(* CODESYS project PRO_JSON 1.0.0.13.library
   Version: 1.0.0.13
   Title: PRO JSON
   Author: TVM
   DocFormat: reStructuredText
   Placeholder: PRO_JSON
   Company: Pro Electric
   DefaultNamespace: PRO_JSON

Project tree, tasks and I/O mapping:
  libraries: Standard, 3.5.15.0 (System); StringUtils, 3.5.15.0 (System); SysMem, 3.5.12.0 (System)
  00000000-0000-0000-0000-000000000000|D:\Dropbox\Pro Electric\Codesys Libraries Development\Pro Electric\COPYING.txt
  00000000-0000-0000-0000-000000000000|D:\Dropbox\Pro Electric\Codesys Libraries Development\Pro Electric\GPL COPYRIGHT.txt
  COPYING
  Data Types/
    data type ASCII
    data type JSONNAMEVALUE
    data type JSONVALUETYPE
    function block JSONVAR [ST]: AsString, Boolean, CharString, FB_Init, Integer, Null, Number, ApplicationLevel, Size, ValueType, VarName, AsDateTime, Init
    data type JSONVARNAME
  Examples/
    data type EXAMPLEJSONSTRUCT
    data type EXAMPLEJSONSTRUCT_1
    program ExampleJSON_PRG [ST]
    function block EXAMPLE_FB [ST]
    program Test_ArrayOfStruct_PRG [ST]
    program Test_Array_PRG [ST]
    program Test_NestedStruct_PRG [ST]
    program Test_SingleVar_PRG [ST]
    program Test_Struct_PRG [ST]
    data type ARRAYOFSTRUCT
    data type JSONSTRUCT
    data type JSONSTRUCT_1
  Functions/
    function CLEANSTRING [ST]
    function ISBOOLEAN [ST]
    function ISNUMBER [ST]
    function block JSON_TO_STRUCT [ST]: CloseArray, CloseObject, Comma, ErrorHandler, Name, OpenArray, OpenObject, Value
    function REAL_TO_STRING_X [ST]
    function SPLIT_VARNAME [ST]
    function block STRUCT_TO_JSON [ST]: CloseArray, CloseObject, CreateArray, CreateName, CreateObject, CreateValue, ErrorHandler, Init
    function ISINTEGER [ST]
    function JSONVALUE_TO_STRING [ST]
    function STRING_TO_JSONVALUE [ST]
    function MATCH_NAMES [ST]
  GPL_COPYRIGHT
  global variables GPL_JSON
  program Notes [ST]
*)

// Data Types/ASCII
(*
| Author: Tim Van Meppelen, Pro Electric Inc.
| timv@proelectric.com
| Date: Nov 2, 2018
| enumeration of all ascii characters
*)
TYPE ASCII :
//ASCII table character definitions
(
	NULL:=			0,
 	SOH:= 			1,
 	STX:=           2,
 	ETX:=           3,
 	EOT:=           4,
 	ENQ:=           5,
 	ACK:=           6,
 	BEL:=           7,
 	BS:=            8,
 	HT:=            9,
 	LF:=            10,
 	VT:=            11,
 	FF:=            12,
 	CR:=            13,
 	SO:=            14,
 	SI:=            15,
 	DLE:=           16,
 	DC1:=           17,
 	DC2:=           18,
 	DC3:=           19,
 	DC4:=           20,
 	NAK:=           21,
 	SYN:=           22,
 	ETB:=           23,
 	CAN:=           24,
 	EM:=            25,
 	SUB_:=			26,
 	ESC:=           27,
 	FS:=            28,
 	GS:=            29,
 	RS:=            30,
 	US:=            31,
	SPACE:=			32,
	BANG:=			33,
	DOUBLE_QUOTE:=	34,
	HASH:=			35,
	DOLLAR:=		36,
	PERCENT:=		37,
	AMPERSAND:=		38,
	SINGLE_QUOTE:=	39,
	OPEN_PAREN:=	40,
	CLOSE_PAREN:=	41,
	STAR:=			42,
	PLUS:=			43,
	COMMA:=			44,
	MINUS:=			45,
	DOT:=			46,	
	SLASH:=			47,
	NUMBER_0:=		48,
	NUMBER_1:=		49,
	NUMBER_2:=		50,
	NUMBER_3:=		51,
	NUMBER_4:=		52,
	NUMBER_5:=		53,
	NUMBER_6:=		54,
	NUMBER_7:=		55,
	NUMBER_8:=		56,
	NUMBER_9:=		57,
	COLON:=			58,	
	SEMICOLON:=		59,
	LESS_THAN:=		60,
	EQUALS:=		61,
	GREATER_THAN:=	62,
	QUESTION:=		63,
	AT_SIGN:=		64,
	UPPERCASE_A:=	65,
	UPPERCASE_B:=	66,
	UPPERCASE_C:=	67,
	UPPERCASE_D:=	68,
	UPPERCASE_E:=	69,
	UPPERCASE_F:=	70,
	UPPERCASE_G:=	71,
	UPPERCASE_H:=	72,
	UPPERCASE_I:=	73,
	UPPERCASE_J:=	74,
	UPPERCASE_K:=	75,
	UPPERCASE_L:=	76,
	UPPERCASE_M:=	77,
	UPPERCASE_N:=	78,
	UPPERCASE_O:=	79,
	UPPERCASE_P:=	80,
	UPPERCASE_Q:=	81,
	UPPERCASE_R:=	82,
	UPPERCASE_S:=	83,
	UPPERCASE_T:=	84,
	UPPERCASE_U:=	85,
	UPPERCASE_V:=	86,
	UPPERCASE_W:=	87,
	UPPERCASE_X:=	88,
	UPPERCASE_Y:=	89,
	UPPERCASE_Z:=	90,
	OPEN_BRACKET:=	91,
	BACKSLASH:=		92,
	CLOSE_BRACKET:=	93,	
	CARET:=			94,
	UNDERSCORE:=	95,
	BACKQUOTE:=		96,
	LOWERCASE_A:=	97,
	LOWERCASE_B:=	98,
	LOWERCASE_C:=	99,
	LOWERCASE_D:=	100,
	LOWERCASE_E:=	101,
	LOWERCASE_F:=	102,
	LOWERCASE_G:=	103,
	LOWERCASE_H:=	104,
	LOWERCASE_I:=	105,
	LOWERCASE_J:=	106,
	LOWERCASE_K:=	107,
	LOWERCASE_L:=	108,
	LOWERCASE_M:=	109,
	LOWERCASE_N:=	110,
	LOWERCASE_O:=	111,
	LOWERCASE_P:=	112,
	LOWERCASE_Q:=	113,
	LOWERCASE_R:=	114,
	LOWERCASE_S:=	115,
	LOWERCASE_T:=	116,
	LOWERCASE_U:=	117,
	LOWERCASE_V:=	118,
	LOWERCASE_W:=	119,
	LOWERCASE_X:=	120,
	LOWERCASE_Y:=	121,
	LOWERCASE_Z:=	122,
	OPEN_BRACE:=	123,
	PIPE:=			124,
	CLOSE_BRACE:=	125,
	TILDE:=			126,
	DEL:=			127
) BYTE;
END_TYPE

// Data Types/JSONNAMEVALUE
(*
| Author: Tim Van Meppelen, Pro Electric Inc.
| timv@proelectric.com
| Date: Nov 2, 2018
| name : value pair
*)
TYPE JSONNAMEVALUE :
STRUCT
	Name:			STRING(GPL_JSON.MAX_NAME_SIZE);		//name of the object at this level
	Value:			STRING(GPL_JSON.MAX_VALUE_SIZE);	//value of the object at this level
	ArrayIndex:		UINT;	//array index of the object at this level
	IsArray:		BOOL;
END_STRUCT
END_TYPE

// Data Types/JSONVALUETYPE
(*
| Author: Tim Van Meppelen, Pro Electric Inc.
| timv@proelectric.com
| Date: Nov 2, 2018
| enumeration of all json types
| NOTE: JSON standard is somewhat ambiguous with number types, so integer and floating point numbers are separate types in this library
*)
TYPE JSONVALUETYPE :
(
	json_string,	//local var is type STRING
	json_number,	//local var is REAL
	json_integer,	//local var is DINT
	json_boolean,	//local var is BOOL
	json_null,		//local var is type null
	json_array,		//object is an array
	json_object		//object is another object (nested objects)
);
END_TYPE

// Data Types/JSONVARNAME
(*
| Author: Tim Van Meppelen, Pro Electric Inc.
| timv@proelectric.com
| Date: Nov 2, 2018
| variable name structure, used with JSONVAR
*)
TYPE JSONVARNAME :
STRUCT
	Name:			STRING(GPL_JSON.MAX_NAME_SIZE);	//name of this variable or object
	ArrayIndex:		UINT;			//array index of the object at this level
	NewObject:		BOOL;			//first variable of a new object
	EndObject:		BOOL;			//last variable of an object
	NewArray:		BOOL;			//first variable of a new array
	EndArray:		BOOL;			//last variable of an array
END_STRUCT
END_TYPE

// Examples/EXAMPLEJSONSTRUCT
(*
| Author: Tim Van Meppelen, Pro Electric Inc.
| timv@proelectric.com
| Date: Jan 31, 2020
| example of a struct of json variables
*)
TYPE EXAMPLEJSONSTRUCT :
STRUCT
	var1:		JSONVAR;
	var2:		JSONVAR;
	var3:		JSONVAR;
	obj:		EXAMPLEJSONSTRUCT_1;
	arrayobj:	ARRAY[1..3] OF JSONVAR;
END_STRUCT
END_TYPE

// Examples/EXAMPLEJSONSTRUCT_1
(*
| Author: Tim Van Meppelen, Pro Electric Inc.
| timv@proelectric.com
| Date: Jan 31, 2020
| example of a struct of json variables
*)
TYPE EXAMPLEJSONSTRUCT_1 :
STRUCT
	var4:		JSONVAR;
	var5:		JSONVAR;
	var6:		JSONVAR;
	var7:		ARRAY[1..3] OF JSONVAR;
END_STRUCT
END_TYPE

// Examples/ARRAYOFSTRUCT
TYPE ARRAYOFSTRUCT :
STRUCT
	arr:			ARRAY[1..4] OF  JSONSTRUCT;
END_STRUCT
END_TYPE

// Examples/JSONSTRUCT
TYPE JSONSTRUCT :
STRUCT
	obj1:		JSONVAR;
	_obj2:		JSONVAR;
	obj3:		JSONVAR;
END_STRUCT
END_TYPE

// Examples/JSONSTRUCT_1
TYPE JSONSTRUCT_1 :
STRUCT
	obj1:		JSONVAR;
	obj2:		JSONVAR;
	obj3:		JSONVAR;
	nest:		JSONSTRUCT;
END_STRUCT
END_TYPE

// GPL_JSON
(*
| Author: Tim Van Meppelen, Pro Electric Inc.
| timv@proelectric.com
| Date: June 26, 2018
| Parameter list that contains limits on size of strings, arrays, etc.  Most of these variables are simply
| to limit memory usage, so they can be increased or decreased to suit the local application and controller
*)
{attribute 'qualified_only'}
VAR_GLOBAL CONSTANT
	MAX_LEVELS:					UINT:= 15;		//maximum number of nested object levels
	MAX_NAME_SIZE:				UINT:= 40;		//max string length of JSON name
	MAX_VALUE_SIZE:				UINT:= 20;		//max value size in bytes (all values are this size in memory)
	MAX_VAR_NAME:				UINT:= 200;		//maximum length of full variable name with path
	MAX_VARS:					UINT:= 1500;	//maximum number of variables in the local structure
	MAX_EXECUTION_TIME:			TIME:= T#50MS;	//maximum time for a single scan of the JSON_TO_STRUCT function block
	MAX_JSON_STRING:			UINT:= 20000;	//maximum allowable size of JSON string
	NEWLINE:					STRING(2):= '$0D$0A';	//formatting string for new line
	INDENT:						STRING(1):= '$T';	//formatting string for indentation
	IGNORE_LEADING_CHAR:		STRING(1):= '_';		//ignore first character in variable names
END_VAR

// Notes
(*
| Author: Tim Van Meppelen, Pro Electric Inc.
| timv@proelectric.com
| Date: Nov 2, 2018
| 
| Tested with 200mS cyclic task, GPL_JSON.MAX_EXECUTION_TIME=50mS
| Depending on the application and speed of the controller, these values could be changed. 
| Be aware of how much cycle time is being taken when using multiple function blocks.
| Each function block will limit its time to GPL_JSON.MAX_EXECUTION_TIME, but multiple function blocks 
| could take up more than that.  This is on the list of things that could be improved. 
| 
| JSONVAR
| FB_Init will fill in information about the variable name and structure in VarNameArray
| variable type and size are automatically determined when a value is set, either:
| 	-with the set accessor of the AsString Property, which will make a guess at the type, based on the value
| 	-with any of the set accessors of the CharString, Boolean, Integer, Number, or Null properties
| variable name is set automatically in FB_Init
| 	-variable name is the JSON name
| 	-JSON allows some object names that are not valid variable names in IEC61131, for example "type", 
| 	"3h", etc.  Workaround is to put an underscore at the beginning of the variable name.  This will
| 	match in JSON_TO_STRUCT, and STRUCT_TO_JSON will create a name without the leading underscore
| 	
| JSON_TO_STRUCT
| convert a JSON string into a local structure of JSONVAR
| Long strings can take several seconds--for example, I have tested with a string of 20kB length, and the 
| parse time is about 4 seconds.  Ensuring that the local variable structure is designed to be as close as 
| possible to the expected order of variables in the JSON string will decrease parsing time, the search loop 
| always starts with the next local variable and loops around until a match is found.
| 
| STRUCT_TO_JSON
| convert a local structure of JSONVAR to a JSON string
| .Format input will create indenting and new lines, useful for writing to a file TO DO: not tested yet
| 
| GPL_JSON
| Parameter list that contains limits on size of strings, arrays, etc.  Most of these variables are simply
| to limit memory usage, so they can be increased or decreased to suit the local application and controller
|
| NEW IDEAS
| -speed up
| -JSON_STRINGIFY function that can be called multiple times to create a JSON string from key and value string inputs
| 	-would create JSON on the fly without having to define a JSONVAR structure
| 	-could be useful for small strings, HTTP server responses, etc
|	-JSONVAR.SetValue() method with ANY input might be a more convenient way to set variable values than using properties
*)
PROGRAM Notes

END_PROGRAM

// Data Types/JSONVAR
(*
| Author: Tim Van Meppelen, Pro Electric Inc.
| timv@proelectric.com
| Date: Nov 2, 2018
| local JSON variables
| 
| for use with JSON_TO_STRUCT, STRUCT_TO_JSON
| variable type and size are automatically determined when a value is set, either:
| 
| - with the set accessor of the AsString Property, which will make a guess at the type, based on the value
| - with any of the set accessors of the CharString, Boolean, Integer, Number, or Null properties
| 
| | variable name is set automatically in FB_Init:
| 
| - variable name is the JSON name
| - JSON allows some object names that are not valid variable names in IEC61131, for example "type", "3h", etc.  
| Workaround is to put a character (default: underscore) at the beginning of the variable name.  This will match in JSON_TO_STRUCT, 
| and STRUCT_TO_JSON will create a name without the leading underscore.  Character can be changed in GPL_JSON.IGNORE_LEADING_CHAR
*)
{attribute 'pack_mode' := '4'}
{attribute 'reflection'}
{attribute 'symbol' := 'none'}
FUNCTION_BLOCK JSONVAR
VAR_INPUT
	Names:			ARRAY[1..GPL_JSON.MAX_LEVELS] OF JSONVARNAME;	//variable path as an array. [1] is variable name, [2..x] are higher level structures	
END_VAR
VAR
	{attribute 'instance-path'}{attribute 'noinit'}
	{attribute 'hide'}_VarNameFull: 		STRING(GPL_JSON.MAX_VAR_NAME);   				//JSON name uses the variable name
	{attribute 'hide'}_ValueType:			JSONVALUETYPE:= JSONVALUETYPE.json_null;		//type of variable contained in the value field, also implicity defines size of local var
	{attribute 'hide'}_InternalValue:		ARRAY[1..GPL_JSON.MAX_VALUE_SIZE+1] OF BYTE;	//value stored internally as an array of bytes
	{attribute 'hide'}_Size:				UINT;										//size of internal value in bytes, automatically determined when any of the type properties are set
	{attribute 'hide'}_ApplicationLevel:	INT;										//array position which points to the application
	{attribute 'hide'}_InitDone:			BOOL;										//save if this element/ struc ... was initialisised
END_VAR
VAR_OUTPUT
	{attribute 'symbol' := 'read'}HMIVarAsString:	STRING(GPL_JSON.MAX_VALUE_SIZE); //this output is updated every time AsString property is set, for use with external HMI through sumbol configuration
END_VAR
VAR_STAT
	{attribute 'hide'}PrevApplicationLevel:	REFERENCE TO INT;		//highest variable name in previous variable
	{attribute 'hide'}PrevNameArray:		REFERENCE TO ARRAY[1..GPL_JSON.MAX_LEVELS] OF JSONVARNAME;//path of the previous variable
END_VAR

{attribute 'monitoring':='call'}PROPERTY AsString : STRING(GPL_JSON.MAX_VALUE_SIZE)
GET
(*
| Author: Tim Van Meppelen, Pro Electric Inc.
| timv@proelectric.com
| Date: Nov 2, 2018
| get the variable value as a string
*)
AsString:= JSONVALUE_TO_STRING(THIS);
END_GET
SET
(*
| Author: Tim Van Meppelen, Pro Electric Inc.
| timv@proelectric.com
| Date: Nov 2, 2018
| set the variable value as a string
*)
VAR

END_VAR
STRING_TO_JSONVALUE(
	In_String:= AsString,
	Out_JSON:= THIS
);

HMIVarAsString:= AsString;
END_SET
END_PROPERTY

{attribute 'monitoring':='call'}PROPERTY Boolean : BOOL
GET
(*
| Author: Tim Van Meppelen, Pro Electric Inc.
| timv@proelectric.com
| Date: Nov 2, 2018
| get a a boolean variable from the internal value
*)
Boolean:= BYTE_TO_BOOL(_InternalValue[1]);
END_GET
SET
(*
| Author: Tim Van Meppelen, Pro Electric Inc.
| timv@proelectric.com
| Date: Nov 2, 2018
| this is a boolean variable, copy to internal value and set type and size
*)
_ValueType:= JSONVALUETYPE.json_boolean;
_Size:= 1;

//clear memory
SysMemSet(
	pDest:= ADR(_InternalValue), 
	udiValue:= 0, 
	udiCount:= SIZEOF(_InternalValue)
);

//put data into internal value
SysMemCpy(
	pDest:= ADR(_InternalValue), 
	pSrc:= ADR(Boolean), 
	udiCount:= _Size
);
END_SET
END_PROPERTY

{attribute 'monitoring':='call'}PROPERTY CharString : STRING(GPL_JSON.MAX_VALUE_SIZE)
GET
(*
| Author: Tim Van Meppelen, Pro Electric Inc.
| timv@proelectric.com
| Date: Nov 2, 2018
| get a string variable from the internal value
*)
VAR
	TempVar:		STRING(255);
END_VAR
SysMemCpy(
	pDest:= ADR(TempVar), 
	pSrc:= ADR(_InternalValue), 
	udiCount:= _Size+1
);
CharString:= TempVar;
END_GET
SET
(*
| Author: Tim Van Meppelen, Pro Electric Inc.
| timv@proelectric.com
| Date: Nov 2, 2018
| this is a string variable, copy to internal value and set type and size
*)
_ValueType:= JSONVALUETYPE.json_string;
_Size:= INT_TO_UINT(LEN(CharString));

//clear memory
SysMemSet(
	pDest:= ADR(_InternalValue), 
	udiValue:= 0, 
	udiCount:= SIZEOF(_InternalValue)
);

//put data into internal value
SysMemCpy(
	pDest:= ADR(_InternalValue), 
	pSrc:= ADR(CharString), 
	udiCount:= _Size+1
);
END_SET
END_PROPERTY

(*
| Author: Tim Van Meppelen, Pro Electric Inc.
| timv@proelectric.com
| Date: Nov 2, 2018
| split the variable path into an array, and determine some object characteristics
| example variable path: 'Test_M241.Test_M241.Application.TestJSON_PRG.TestStruct.var1'
*)
METHOD FB_Init : BOOL
VAR_INPUT
  bInitRetains : 		BOOL; // TRUE: the retain variables are initialized (reset warm / reset cold)
  bInCopyCode : 		BOOL;  // TRUE: the instance will be copied to the copy code afterward (online change)
END_VAR

VAR
	ArrayPosition:		UINT:= GPL_JSON.MAX_LEVELS;
	NameStringPtr:		POINTER TO ARRAY[1..GPL_JSON.MAX_VAR_NAME] OF BYTE;
	StringIndex:		INT;
	VarNameBegin:		INT;
	VarNameEnd:			INT;
	VarNameIndex:		INT;
	offset:				INT;
	startarraystr:		INT;
	endarraystr:		INT;
	varlevelindex:		INT;
	prevvarlevelindex:	INT;
	stoploop:			INT;
	startloop:			INT;
	FirstVar:			BOOL;
	i:					INT;
END_VAR
//====================GET VARIABLE NAME INTO AN ARRAY====================
NameStringPtr:= ADR(_VarNameFull);
StringIndex:= LEN(_VarNameFull);
VarNameEnd:= StringIndex;
VarNameIndex:= 1;

WHILE (StringIndex > 0) DO
	IF (NameStringPtr^[StringIndex] = ASCII.DOT) THEN
	//found a "." character
		VarNameBegin:= StringIndex + 1;
		
		(*
		//clear array string  TO DO:  IS THIS NECESSARY?
		Sysmem.SysMemSet(
			pDest:= ADR(Names[VarNameIndex]), 
			udiValue:= 0, 
			udiCount:= GPL_JSON.MAX_NAME_SIZE
		);
		*)
		//copy string between VarNameBegin and VarNameEnd
		SysMem.SysMemCpy(
			pDest:= ADR(Names[VarNameIndex]), 
			pSrc:= ADR(NameStringPtr^[VarNameBegin]), 
			udiCount:= INT_TO_UDINT((VarNameEnd - VarNameBegin)+1)
		);

		//check if this is an array, if yes then remove the array index from the variable name
		startarraystr:= FIND(STR1:= Names[VarNameIndex].Name, STR2:= '[');
		endarraystr:= FIND(STR1:= Names[VarNameIndex].Name, STR2:= ']');
		IF (startarraystr <> 0) AND (endarraystr <> 0) THEN
			Names[VarNameIndex].ArrayIndex:= STRING_TO_UINT(MID(
				STR:= Names[VarNameIndex].Name, 
				LEN:= endarraystr-startarraystr-1, 
				POS:= startarraystr+1
			));
			Names[VarNameIndex].Name:= DELETE(
				STR:= Names[VarNameIndex].Name, 
				LEN:= endarraystr-startarraystr+1, 
				POS:= startarraystr
			);
		END_IF
		
		IF (Names[VarNameIndex].Name = 'Application') THEN
		//was this the application level?	
			_ApplicationLevel:= VarNameIndex;
			EXIT;
		END_IF
	
		VarNameIndex:= VarNameIndex + 1;
		VarNameEnd:= VarNameBegin - 2;	//end of the next variable name is known, store for next loop			
		StringIndex:= VarNameBegin - 2;
	ELSE
		StringIndex:= StringIndex - 1;
	END_IF
END_WHILE

//====================JSON OBJECT CHARACTERISTICS====================
(*VAR_STAT PrevApplicationLevel and PrevNameArray are references to the last JSONVAR variable
that was worked on.  This would be the previous variable in a structure or array, but
could also be a variable contained in a completely different JSON structure.
Because it is not possible to reference the next variable in a structure (because
its FB_Init() method has not run yet), the characteristics of the last variable 
in a structure are set in the STRUCT_TO_JSON function block.*)

//First variable of a structure
IF __ISVALIDREF(PrevNameArray) THEN
//there is a valid reference to a previous variable, check the previous object
	;	(*NOTE:
		I don't know if it is possible to determine whether this variable is the beginning of a new structure
		or not.  There are so many possible combinations of variables, function blocks, and structures, and the only 
		information this program has to work with is the string which contains the path.  This string only contains
		names, and does not give any information about the type of variable, or which other variables are included
		This functionality is now contained in STRUCT_TO_JSON, which is able to determine the first and last
		variables in a structure.  There's nothing really wrong with this, except that it makes the code a bit more
		difficult to understand, as there's two locations that work on variable characteristics.*)
ELSE
//there is no valid reference to a previous variable, indicating that this is the first time FB_Init has run anywhere in the application
//therefore, this is the first variable of a new JSON object
	FirstVar:= TRUE;
END_IF

IF FirstVar THEN
//first variable of a new structure
	FOR varlevelindex:= 1 TO _ApplicationLevel-2 DO
		//every level of the first variable could be either a new object or a new array
		IF (Names[varlevelindex].ArrayIndex = 1) THEN
		//new array
			Names[varlevelindex].NewArray:= TRUE;	
		ELSIF (varlevelindex > 1) THEN
		//new object
			Names[varlevelindex].NewObject:= TRUE;
		END_IF			
	END_FOR
ELSE	
//not the first variable of a new structure
	offset:= _ApplicationLevel - PrevApplicationLevel;	//check if the variable names have shifted up or down
	IF (offset < 0) THEN
	//objects shifted down
		stoploop:= PrevApplicationLevel - 1;
		startloop:= 1;
	ELSE
	//no shift, or shift up
		stoploop:= _ApplicationLevel - 1;
		startloop:= offset + 1;
	END_IF
	FOR varlevelindex:= startloop TO stoploop DO
		prevvarlevelindex:= varlevelindex - offset;
		
		//====================End previous array====================
		IF (offset < 0) AND (varlevelindex = 1) THEN
		//if objects have shifted down, then varlevelindex-offset will never point to PrevNameArray[1]
		//the previous variable might need an array closed
			IF (PrevNameArray[1].ArrayIndex > 0) THEN
			//end array
				PrevNameArray[1].EndArray:= TRUE;
			END_IF	
		END_IF

		IF (PrevNameArray[prevvarlevelindex].ArrayIndex > 0) AND (Names[varlevelindex].Name <> PrevNameArray[prevvarlevelindex].Name) THEN
			PrevNameArray[prevvarlevelindex].EndArray:= TRUE;
		END_IF	
		
		//====================End previous object====================
		IF ((varlevelindex-offset) > 1) AND ((Names[varlevelindex].Name <> PrevNameArray[prevvarlevelindex].Name) OR (Names[varlevelindex].ArrayIndex <> PrevNameArray[prevvarlevelindex].ArrayIndex)) THEN
			PrevNameArray[prevvarlevelindex].EndObject:= TRUE;	//close previous object	
		END_IF	
		
		//====================New array====================
		IF (Names[varlevelindex].ArrayIndex = 1) AND (PrevNameArray[prevvarlevelindex].ArrayIndex = 0) THEN
			Names[varlevelindex].NewArray:= TRUE;				
		END_IF	
	
		//====================New object====================
		IF (varlevelindex > 1) AND ((NOT Names[varlevelindex].NewArray) AND (Names[varlevelindex].Name <> PrevNameArray[prevvarlevelindex].Name) OR (Names[varlevelindex].ArrayIndex <> PrevNameArray[prevvarlevelindex].ArrayIndex)) THEN
			Names[varlevelindex].NewObject:= TRUE;	//new object at this level	
		END_IF	
	END_FOR

END_IF

//set a reference to some variables for the next JSON variable
PrevNameArray REF= Names;
PrevApplicationLevel REF= _ApplicationLevel;
END_METHOD

{attribute 'monitoring':='call'}PROPERTY Integer : DINT
GET
(*
| Author: Tim Van Meppelen, Pro Electric Inc.
| timv@proelectric.com
| Date: Mar 2, 2020
| get an integer variable from the internal value
| Note: .Integer and .Number are the only two properties which do type conversion on the fly because 
| the JSON standard doesn't strictly define the difference between an integer and a floating point number
*)
VAR
	tempDINT:	DINT;
	tempREAL:	REAL;
END_VAR
CASE _ValueType OF
JSONVALUETYPE.json_number:
//internal value was stored as floating point, convert to integer
	SysMemCpy(
		pDest:= ADR(tempREAL), 
		pSrc:= ADR(_InternalValue), 
		udiCount:= 4
	);
	Integer:= REAL_TO_DINT(tempREAL);		
JSONVALUETYPE.json_integer:
//internal value was stored as integer, get the value
	SysMemCpy(
		pDest:= ADR(tempDINT), 
		pSrc:= ADR(_InternalValue), 
		udiCount:= 4
	);
	Integer:= tempDINT;
END_CASE
END_GET
SET
(*
| Author: Tim Van Meppelen, Pro Electric Inc.
| timv@proelectric.com
| Date: Nov 2, 2018
| this is a integer variable, copy to internal value and set type and size
*)
VAR
	TempVar:		DINT;
END_VAR
_ValueType:= JSONVALUETYPE.json_integer;
_Size:= 4;

//clear memory
SysMemSet(
	pDest:= ADR(_InternalValue), 
	udiValue:= 0, 
	udiCount:= SIZEOF(_InternalValue)
);

TempVar:= Integer;

//put data into internal value
SysMemCpy(
	pDest:= ADR(_InternalValue), 
	pSrc:= ADR(TempVar), 
	udiCount:= _Size
);
END_SET
END_PROPERTY

{attribute 'monitoring':='call'}PROPERTY Null : STRING(4)
GET
(*
| Author: Tim Van Meppelen, Pro Electric Inc.
| timv@proelectric.com
| Date: Nov 2, 2018
| get a null value (returned as a string, as IEC61131 has no way to represent a null value)
*)
Null:= 'null';
END_GET
SET
(*
| Author: Tim Van Meppelen, Pro Electric Inc.
| timv@proelectric.com
| Date: Nov 2, 2018
| this is a null variable, set type and size
*)
_ValueType:= JSONVALUETYPE.json_null;
_Size:= 4;
END_SET
END_PROPERTY

{attribute 'monitoring':='call'}PROPERTY Number : REAL
GET
(*
| Author: Tim Van Meppelen, Pro Electric Inc.
| timv@proelectric.com
| Date: Mar 2, 2020
| get a floating point variable from the internal value
| Note: .Integer and .Number are the only two properties which do type conversion on the fly because 
| the JSON standard doesn't strictly define the difference between an integer and a floating point number
*)
VAR
	tempDINT:	DINT;
	tempREAL:	REAL;
END_VAR
CASE _ValueType OF
JSONVALUETYPE.json_integer:
//internal value was stored as integer, convert to floating point
	SysMemCpy(
		pDest:= ADR(tempDINT), 
		pSrc:= ADR(_InternalValue), 
		udiCount:= 4
	);
	Number:= DINT_TO_REAL(tempDINT);	
	
JSONVALUETYPE.json_number:
//internal value was stored as floating point, get value
	SysMemCpy(
		pDest:= ADR(tempREAL), 
		pSrc:= ADR(_InternalValue), 
		udiCount:= 4
	);
	Number:= tempREAL;	
END_CASE
END_GET
SET
(*
| Author: Tim Van Meppelen, Pro Electric Inc.
| timv@proelectric.com
| Date: Nov 2, 2018
| this is a floating point variable, copy to internal value and set type and size
*)
_ValueType:= JSONVALUETYPE.json_number;
_Size:= 4;

//clear memory
SysMemSet(
	pDest:= ADR(_InternalValue), 
	udiValue:= 0, 
	udiCount:= SIZEOF(_InternalValue)
);

//put data into internal value
SysMemCpy(
	pDest:= ADR(_InternalValue), 
	pSrc:= ADR(Number), 
	udiCount:= _Size
);
END_SET
END_PROPERTY

{attribute 'monitoring':='call'}PROPERTY ApplicationLevel : INT
GET
(*
| Author: Tim Van Meppelen, Pro Electric Inc.
| timv@proelectric.com
| Date: Nov 2, 2018
| array position which points to the application level
*)
ApplicationLevel:= _ApplicationLevel;
END_GET
END_PROPERTY

{attribute 'monitoring':='call'}PROPERTY Size : UINT
GET
(*
| Author: Tim Van Meppelen, Pro Electric Inc.
| timv@proelectric.com
| Date: Nov 2, 2018
| size of internal value in bytes, automatically determined when any of the type properties are set
*)
Size:= _Size;
END_GET
END_PROPERTY

{attribute 'monitoring':='call'}PROPERTY ValueType : JSONVALUETYPE
GET
(*
| Author: Tim Van Meppelen, Pro Electric Inc.
| timv@proelectric.com
| Date: Nov 2, 2018
| type of variable contained in the value field, also implicity defines size of local var
*)
ValueType:= _ValueType;
END_GET
SET
_ValueType:= ValueType;
END_SET
END_PROPERTY

{attribute 'monitoring':='call'}PROPERTY VarName : STRING(GPL_JSON.MAX_VAR_NAME)
GET
(*
| Author: Tim Van Meppelen, Pro Electric Inc.
| timv@proelectric.com
| Date: Sept 16, 2019
| get the name of the variable as a string, ie.
| 'Test_M241.Test_M241.Application.TestJSON_PRG.TestStruct.var1'
*)
VarName:= _VarNameFull;
END_GET
SET
(*
| Author: Tim Van Meppelen, Pro Electric Inc.
| timv@proelectric.com
| Date: Sept 16, 2019
| 
| Manually set JSON variable name to something other than it's automatically generated name.  This should only 
| be used when the JSON string could have a changing variable name at runtime, ie. the variable name is a date 
| or a counter.  Normally, the JSON variable name is the same as the PLC variable name
| NOTE:  this cannot change the number of levels of a nested object, it is assumed that the basic structure
| remains the same, and only the names are changing
| 
| example created by FB_Init:
| _VarNameFull   'Test_M241.Application.TestJSON_PRG.TestStruct.var1'
| _VarNameArray                 [4]        [3]          [2]     [1]
| _ApplicationLevel = 2
| 
| example after runtime changes
| _VarNameFull   'TestStruct.var1'
| _VarNameArray      [2]     [1]
| _ApplicationLevel = 2
| 
| set as a string ie. 'TestStruct.var1'
| each object inside another object must be changed manually
| higher level object names must be changed in each lower level object
| program level and above are not manually adjustable at runtime ie. 'Test_M241.Application.TestJSON_PRG.'
*)
VAR
	Levels:			UINT;
	i:				INT;
END_VAR
Levels:= SPLIT_VARNAME(VarNameArray:= Names, StringIn:= VarName);

FOR i:= UINT_TO_INT(Levels) TO 1 BY -1 DO 
//recreate the var name string
	IF (i = UINT_TO_INT(Levels)) THEN
		_VarNameFull:= CONCAT(Names[i].Name,'.');
	ELSIF (i = 1) THEN
		_VarNameFull:= CONCAT(_VarNameFull, Names[i].Name);
	ELSE
		_VarNameFull:= CONCAT(_VarNameFull, Names[i].Name);
		_VarNameFull:= CONCAT(_VarNameFull, '.');
	END_IF
END_FOR
END_SET
END_PROPERTY

{attribute 'monitoring':='call'}PROPERTY AsDateTime : DT
GET
(*
| Author: Tim Van Meppelen, Pro Electric Inc.
| timv@proelectric.com
| Date: Mar 2, 2020
| get a numeric JSON variable to a DATE_AND_TIME variable
*)
CASE _ValueType OF
JSONVALUETYPE.json_number:
	AsDateTime:= REAL_TO_DT(THIS^.Number);
JSONVALUETYPE.json_integer:
	AsDateTime:= DINT_TO_DT(THIS^.Integer);
JSONVALUETYPE.json_string:
	AsDateTime:= STRING_TO_DT(THIS^.CharString);
END_CASE
END_GET
SET
(*
| Author: Tim Van Meppelen, Pro Electric Inc.
| timv@proelectric.com
| Date: Mar 2, 2020
| convert the value from DATE_AND_TIME format and set it to whatever type of variable is already configured
*)
VAR
	TempReal:	REAL;
	TempInt:	DINT;
	TempString:	STRING(255);
END_VAR
CASE _ValueType OF
JSONVALUETYPE.json_number:
	TempReal:= DT_TO_REAL(AsDateTime);
	THIS^.Number:= TempReal;
JSONVALUETYPE.json_integer:
	TempInt:= DT_TO_DINT(AsDateTime);
	THIS^.Integer:= TempInt;	
JSONVALUETYPE.json_string:
	TempString:= DT_TO_STRING(AsDateTime);
	THIS^.CharString:= TempString;
END_CASE
END_SET
END_PROPERTY

PROPERTY Init : bool
SET
_InitDone:= Init;
END_SET
GET
Init:= _InitDone;
END_GET
END_PROPERTY

END_FUNCTION_BLOCK

// Functions/JSON_TO_STRUCT
(*
| Author: Tim Van Meppelen, Pro Electric Inc.
| timv@proelectric.com
| Date: Nov 2, 2018
| Last Modified: Jan 4, 2022
| parse JSON string and place the values in a matching local structure of type JSONVAR
*)
FUNCTION_BLOCK JSON_TO_STRUCT
VAR_INPUT
	Execute:			BOOL;		//rising edge triggers parse of JSON string
	Abort:				BOOL;		//rising edge stops parsing of JSON string
	JSONString:			POINTER TO ARRAY[1..GPL_JSON.MAX_JSON_STRING] OF ASCII;	//pointer to JSON string
	JSONStringSize:		UDINT;		//size of string in bytes
	JSONVars:			POINTER TO ARRAY[1..GPL_JSON.MAX_VARS] OF JSONVAR;	//pointer to local structure made up of type JSONVAR
	NumberOfVars:		UDINT;		//number of variables in the local structure or array
END_VAR

VAR_OUTPUT
	Busy:				BOOL;		//busy parsing a string
	Done:				BOOL;		//successfully parsed the whole string with no errors
	Aborted:			BOOL;		//parsing aborted by Abort input
	Error:				BOOL;		//unexpected character detected, string not completely parsed
	ErrorPosition:		UDINT;		//character position where the unexpected character was found
	ParseTime:			TIME;		//time it took to parse the string
END_VAR

VAR
	bufferposition:		UDINT;	//current position in the string
	NameValue:			ARRAY[1..GPL_JSON.MAX_LEVELS] OF JSONNAMEVALUE;	//name:value pairs currently being worked on
	obj_level:			UINT;	//number of nested objects
	name_start:			UDINT;	//index of the beginning of a name
	name_stop:			UDINT;	//index of the end of a name
	value_start:		UDINT;	//index of the beginning of a value
	value_stop:			UDINT;	//index of the end of a value
	findname:			BOOL;	//look for name in configuration array
	foundname:			BOOL;	//found a matching local var
	i:					UDINT;	//loop indexes
	jsonvarindex:		UDINT;
	levelindex:			UINT;
	nameindex:			UINT;
	thisloopstarttime:	TIME;		//time the current loop started
	starttime:			TIME;		//time parsing started
	Execute_TRIG:		R_TRIG;
	Abort_TRIG:			R_TRIG;
	findloop:			UDINT;
	parse:				BOOL;
END_VAR

IF (JSONString = 0) OR (JSONVars = 0) OR (NumberOfVars > GPL_JSON.MAX_VARS) THEN
//Bugfix Jan 4, 2022 suggested by Stefan Dreyer, to eliminate problems with uninitialized pointers	
//can't parse string - increase CPL_JSON.MAX_VARS
	Error:= TRUE;
	RETURN;
END_IF

thisloopstarttime:= TIME();	//store the time of the beginning of this loop	

Execute_TRIG(CLK:= Execute);
Abort_TRIG(CLK:= Abort);
Done:= FALSE;
IF Execute_TRIG.Q THEN
//must see a rising edge on execute to start parsing
	starttime:= TIME();	//store the time of the beginning of execution
	parse:= TRUE;
	bufferposition:= 1;
	Busy:= TRUE;
	Aborted:= FALSE;
	
	Error:= FALSE;
	ErrorPosition:= 0;
	obj_level:= 0;
	FOR i:= 1 TO GPL_JSON.MAX_LEVELS DO
		NameValue[i].Name:= '';
		NameValue[i].Value:= '';
		NameValue[i].IsArray:= FALSE;
		NameValue[i].ArrayIndex:= 0;
	END_FOR
END_IF

IF Abort_TRIG.Q THEN
	Busy:= FALSE;
	Aborted:= TRUE;
	parse:= FALSE;
END_IF

(*====================PARSE JSON STRING====================*)
//parse the input string, and start storing values in NameValue array
WHILE parse DO
	IF (JSONString^[bufferposition] = ASCII.NULL) OR (bufferposition > JSONStringSize) THEN
	//strings are terminated with a null character
	//there might not always be a null character, for example in a network buffer that is stored as an array of bytes
		parse:= FALSE;
		Done:= TRUE;
		Busy:= FALSE;
		ParseTime:= TIME() - starttime;
		RETURN;
	END_IF	

	CASE JSONString^[bufferposition] OF 

	ASCII.DOUBLE_QUOTE:	// " name string
		Name();
		
	ASCII.OPEN_BRACE:// {, beginning of object
		OpenObject();	
		
	ASCII.CLOSE_BRACE:// }, end of object
		CloseObject();
		
	ASCII.OPEN_BRACKET:	// [, beginning of array
		OpenArray();
		
	ASCII.CLOSE_BRACKET:	// ], end of array
		CloseArray();
		
	ASCII.COLON:	// :, separator for name:value pairs
		Value();
		
	ASCII.COMMA:	// , move to next object
		Comma();
	
	ASCII.SOH..ASCII.SPACE:	// skip all control characters, including spaces
		bufferposition:= bufferposition + 1;

	ELSE
	//error, unexpected character
		ErrorHandler();
	END_CASE
	
	(*========================================LOOK FOR NAMES IN LOCAL VARIABLES========================================*)
	IF findname THEN
	//there is at least one valid name:value pair in the NameValue array--check for a match in the Config array, including nested objects
		findname:= FALSE;
		FOR findloop:= 1 TO NumberOfVars DO
		(*loop through all configured objects and look for the name that is currently being worked on in the JSON string
		Local JSON object should be as closely matched to the expected JSON string as possible, to decrease parsing time.  
		This function will eventually find all objects, but it will start looking after the previous found variable, as it 
		is assumed that that's the most likely position for the next variable*)  
			jsonvarindex:= (jsonvarindex MOD NumberOfVars) + 1;
			FOR nameindex:= 1 TO obj_level DO
			//Match name and array index.  Array index will be 0 if the current name:value is not part of an array
				IF MATCH_NAMES(JSONVars^[jsonvarindex].Names[nameindex], NameValue[obj_level-(nameindex-1)]) THEN	
					foundname:= TRUE;	//name in JSON string matches the local variable name
				ELSE
					foundname:= FALSE;	//name in JSON string does not match the local variable name, go to next name
					EXIT;
				END_IF
			END_FOR
			IF foundname THEN
				EXIT;
			END_IF
		END_FOR
	
		(*====================FOUND NAME, WRITE LOCAL VAR====================*)
		IF foundname THEN
		//local var name matches with JSON string name
			foundname:= FALSE;
			JSONVars^[jsonvarindex].AsString:= NameValue[obj_level].Value;	
		END_IF
	END_IF

	IF TIME() >= (thisloopstarttime + GPL_JSON.MAX_EXECUTION_TIME) THEN
	//this function block won't take up more than GPL_JSON.MAX_EXECUTION_TIME on one scan
	//very long strings or files could take too long to parse in one task cycle, and cause a watchdog exception
		RETURN;
	END_IF
END_WHILE

(*
| Author: Tim Van Meppelen, Pro Electric Inc.
| timv@proelectric.com
| Date: Oct 22, 2018
| end of an array
*)
METHOD PRIVATE CloseArray
NameValue[obj_level].IsArray:= FALSE;
NameValue[obj_level].ArrayIndex:= 0;
bufferposition:= bufferposition + 1;
END_METHOD

(*
| Author: Tim Van Meppelen, Pro Electric Inc.
| timv@proelectric.com
| Date: Oct 22, 2018
| end of an object, move down in the object hierarchy
*)
METHOD PRIVATE CloseObject
VAR
	shiftindex:			INT;
END_VAR
NameValue[obj_level].Name:= '';
NameValue[obj_level].Value:= '';
NameValue[obj_level].IsArray:= FALSE;
NameValue[obj_level].ArrayIndex:= 0;
obj_level:= obj_level - 1;
bufferposition:= bufferposition + 1;
END_METHOD

(*
| Author: Tim Van Meppelen, Pro Electric Inc.
| timv@proelectric.com
| Date: Oct 22, 2018
| found a comma, parse an array value, or move on to the next object	
*)
METHOD PRIVATE Comma
IF NameValue[obj_level].IsArray THEN
//if this is an array at the current object level, increment the array index
	NameValue[obj_level].ArrayIndex:= NameValue[obj_level].ArrayIndex + 1;
	Value();
ELSE
	bufferposition:= bufferposition + 1;
END_IF
END_METHOD

(*
| Author: Tim Van Meppelen, Pro Electric Inc.
| timv@proelectric.com
| Date: Oct 22, 2018
| Unexpected or invalid character found, end parsing
*)
METHOD PRIVATE ErrorHandler
parse:= FALSE;
Busy:= FALSE;
Error:= TRUE;
ErrorPosition:= bufferposition;	//return buffer position of unexpected character
END_METHOD

(*
| Author: Tim Van Meppelen, Pro Electric Inc.
| timv@proelectric.com
| Date: Oct 22, 2018
| found the first quote at the beginning of a name string,
| extract the name string and put it into the NameValue array
*)
METHOD PRIVATE Name
VAR
	namestringok:		BOOL;
	j:					UDINT;
END_VAR
name_start:= bufferposition + 1;
FOR j:= name_start TO (name_start+GPL_JSON.MAX_NAME_SIZE) DO
	IF (JSONString^[j] = ASCII.DOUBLE_QUOTE) THEN
	//find the closing quote of a name string
		name_stop:= j - 1;		//name ends at character before quote
		bufferposition:= j + 1;	//next loop can start after the quote
		namestringok:= TRUE;
		EXIT;
	END_IF
END_FOR

IF namestringok THEN
	SysMemSet(
		pDest:= ADR(NameValue[obj_level].Name), 
		udiValue:= 0, 
		udiCount:= SIZEOF(NameValue[obj_level].Name)
	);
	
	SysMemCpy(
		pDest:= ADR(NameValue[obj_level].Name), 
		pSrc:= ADR(JSONString^[name_start]), 
		udiCount:= (name_stop+1 - name_start)
	);
ELSE
	ErrorHandler();
END_IF
END_METHOD

(*
| Author: Tim Van Meppelen, Pro Electric Inc.
| timv@proelectric.com
| Date: Oct 22, 2018
| found the beginning of an array, set array definition at this object level
*)
METHOD PRIVATE OpenArray
VAR_INPUT
END_VAR
NameValue[obj_level].IsArray:= TRUE;
NameValue[obj_level].ArrayIndex:= 1;
bufferposition:= bufferposition + 1;
END_METHOD

(*
| Author: Tim Van Meppelen, Pro Electric Inc.
| timv@proelectric.com
| Date: Oct 22, 2018
| found the beginning of a new object, increment the object level
*)
METHOD PRIVATE OpenObject
VAR
	shiftindex:			INT;
END_VAR
obj_level:= obj_level + 1;	//move up a level in the object hierarchy
bufferposition:= bufferposition + 1;
END_METHOD

(*
| Author: Tim Van Meppelen, Pro Electric Inc.
| timv@proelectric.com
| Date: Oct 22, 2018
| found a ":" character, possible next characters are any combination of the following:
| { begin another object
| [ begin a new array
| " or a number or letter: value found
| after all { and [ are found, and if any were found, the next thing will be a name string
| loop through until a value is found, incrementing obj_level or array definitions as necessary
*)
METHOD PRIVATE Value
VAR
	lookforname:	BOOL;
	j:				UDINT;
	skipnext:		BOOL;
	quotedstring:	BOOL;
END_VAR
bufferposition:= bufferposition + 1;	//start searching after the ":" character

WHILE (bufferposition < JSONStringSize) DO
	CASE JSONString^[bufferposition] OF
		
	ASCII.CR:	// '$r', skip
		bufferposition := bufferposition+1;
		CONTINUE;
	ASCII.LF:	// '$n', skip
		bufferposition := bufferposition+1;
		CONTINUE;
	ASCII.SPACE:	// ' ', skip
		bufferposition := bufferposition+1;
		CONTINUE;
		
	ASCII.OPEN_BRACE:// {, beginning of new object
		OpenObject();	
		lookforname:= TRUE;
	
	ASCII.OPEN_BRACKET:	// [, beginning of new array
		OpenArray();
		
	ELSE
		IF lookforname THEN
		//a new object or array was found, and all nested objects have already been looped through, therefore this buffer position must start a new name
		//there is no value here, so exit this loop, main loop should now continue at the name, and parse its name:value pair
			EXIT;
		END_IF
		
		IF (JSONString^[bufferposition] = ASCII.DOUBLE_QUOTE) THEN
		//value starts with a quote character--quoted string
			value_start:= bufferposition + 1;	//value follows : and "
			quotedstring := TRUE;	
		ELSE
			value_start:= bufferposition;	//value immediately follows :
		END_IF

		FOR j:= value_start TO JSONStringSize DO
			IF skipnext THEN
				skipnext := FALSE;
			ELSIF (JSONString^[j] = ASCII.BACKSLASH)  THEN
				// on backslash, escape the next one
				skipnext := TRUE;
			ELSIF (JSONString^[j] = ASCII.DOUBLE_QUOTE)  THEN
			//end of value is is found at the closing quote
				value_stop:= j - 1;
				bufferposition:= j + 1;	//main loop can resume at the next character after the quote
				EXIT;
			//ELSIF ((JSONString^[j] = ASCII.COMMA) OR (JSONString^[j] = ASCII.CLOSE_BRACE) OR (JSONString^[j] = ASCII.CLOSE_BRACKET)) AND (NOT quotedstring) THEN
			(*bugfix - Dec 8, 2021 Stefan Dryer
			some strings might contain a CR/LF after the value, ahead of the closing bracket*)
			ELSIF ((JSONString^[j] = ASCII.COMMA) OR (JSONString^[j] = ASCII.CLOSE_BRACE) OR (JSONString^[j] = ASCII.CLOSE_BRACKET) OR (JSONString^[j] = ASCII.CR ) OR (JSONString^[j] = ASCII.LF )) AND NOT quotedstring THEN
			//end of value is is found at , or }, or ]
				value_stop:= j - 1;
				bufferposition:= j;	//main loop can resume at the next character after the value
				EXIT;
			END_IF
		END_FOR	
		//clear previous string
		SysMemSet(
			pDest:= ADR(NameValue[obj_level].Value), 
			udiValue:= 0, 
			udiCount:= GPL_JSON.MAX_VALUE_SIZE
		);		
		//copy buffer to temporary value as a string
		SysMemCpy(
			pDest:= ADR(NameValue[obj_level].Value), 
			pSrc:= ADR(JSONString^[value_start]), 
			udiCount:= MIN((value_stop+1) - value_start, GPL_JSON.MAX_VALUE_SIZE-1)
		);
		
		findname:= TRUE;		//there is a name:value pair in the NameValue array, check for a match with a local variable
		EXIT;
	END_CASE
END_WHILE
END_METHOD

END_FUNCTION_BLOCK

// Functions/MATCH_NAMES
(*
| Author: Tim Van Meppelen, Pro Electric Inc.
| timv@proelectric.com
| Date: May 7, 2021
| compare name in JSON string with local variable name
| match when local variable name contains a leading underscore, if present
| JSON allows some object names that are not valid variable names in IEC61131, for example "type", 
| "3h", etc.  Workaround is to put an underscore at the beginning of the variable name.
| this leading underscore can be changed or not used by modifying GPL_JSON.IGNORE_LEADING_CHAR
*)
FUNCTION MATCH_NAMES : BOOL
VAR_INPUT
	Name1:			JSONVARNAME;	//name:value in local value
	Name2:			JSONNAMEVALUE;	//name:value from JSON string
END_VAR
VAR
	LocalVarName:	STRING(GPL_JSON.MAX_NAME_SIZE);	//name stripped of leading underscore, if present
END_VAR

IF (FIND(STR1:= Name1.Name, STR2:= GPL_JSON.IGNORE_LEADING_CHAR) = 1) THEN
//leading character is present, delete it 
	LocalVarName:= DELETE(Name1.Name,1,1);
END_IF

MATCH_NAMES:= ((Name1.Name = Name2.Name OR (Name2.Name = LocalVarName))AND 
				(Name1.ArrayIndex = Name2.ArrayIndex)) ;

END_FUNCTION

// Functions/STRUCT_TO_JSON
(*
| Author: Tim Van Meppelen, Pro Electric Inc.
| timv@proelectric.com
| with thanks to these contributors:
| Stefan Dreyer github.com/stefandreyer
| Wesley Vercoutere
| Date: Nov 2, 2018
| Last Modified: Jan 4, 2022
| create a JSON string from a structure of JSONVAR types
*)
FUNCTION_BLOCK STRUCT_TO_JSON
VAR_INPUT
	Execute:			BOOL;		//rising edge triggers compose of JSON string
	Abort:				BOOL;		//rising edge stops composing a JSON string
	JSONString:			POINTER TO ARRAY[1..GPL_JSON.MAX_JSON_STRING] OF ASCII;	//pointer to JSON string
	JSONStringSize:		UDINT;		//size of string
	JSONVars:			POINTER TO ARRAY[1..GPL_JSON.MAX_VARS] OF JSONVAR;	//pointer to local structure made up of type JSONVAR
	NumberOfVars:		UINT;		//number of variables in the local structure or array
	VariableArraySize:	BOOL;		//don't write array values which are null, resulting in variable array sizes
	{info <'TO DO:  Format input not tested'>}Format:	BOOL;		//add white space and indenting to the resulting string
	MaxLevel:			INT;		//max level at which to create objects
	(*by default, STRUCT_TO_JSON will create variables starting at (Application level - 2).
	This will work for most variables and structures defined in a program.  If your variable
	or structure is contained inside a function block, or nested in function blocks, it may
	be necessary to set MaxLevel to restrict creating JSON after a certain level
	MaxLevel examples:
	Device: 4, Application: 3, Program: 2, Variable: 1
	Device.Application.TestJSON_PRG.var1, default {"var1":"value"}
	Device.Application.TestJSON_PRG.var1, set MaxLevel=2 to get {TestJSON_PRG:{"var1":"value"}}
	
	Device: 5, Application: 4, Program: 3, Function Block: 2, Variable: 1
	Device.Application.TestJSON_PRG.Test_FB.var1, set MaxLevel=1 to get {"var1":"value"}
	Device.Application.TestJSON_PRG.Test_FB.var1, set MaxLevel=2 to get {Test_FB:{"var1":"value"}}
	Device.Application.TestJSON_PRG.Test_FB.var1, set MaxLevel=3 to get {TestJSON_PRG:{Test_FB:{"var1":"value"}}} 
	*)
END_VAR

VAR_OUTPUT
	Busy:				BOOL;		//busy composing a string
	Done:				BOOL;		//successfully composed the whole string with no errors
	Aborted:			BOOL;		//compose aborted by Abort input
	Error:				BOOL;		//unexpected character detected, string not completely composed
	ErrorPosition:		UDINT;		//index of local object at which composing stopped
	ComposeTime:		TIME;		//time it took to compose the string
END_VAR

VAR
	bufferposition:		UDINT;	//current position in the string
	jsonvarindex:		UDINT;
	compose:			BOOL;	
	objectstr:			STRING(255);	//string created by current variable
	names:				ARRAY[1..GPL_JSON.MAX_LEVELS] OF JSONVARNAME;	//helper variable for names array property
	namesindex:			INT;
	i:					UINT;
	
	Execute_TRIG:		R_TRIG;
	Abort_TRIG:			R_TRIG;
	thisloopstarttime:	TIME;		//time the current loop started
	starttime:			TIME;		//time composing started
	maxlevelindex:		INT;
	closeLevel: 		INT;
	objectLevel: 		INT;
	inArray: 			BOOL;
	lastindex:			UDINT;
	InitDn:				BOOL;
END_VAR

IF (JSONString = 0) OR (JSONVars = 0) OR (NumberOfVars > GPL_JSON.MAX_VARS) THEN
//Bugfix Jan 4, 2022 suggested by Stefan Dreyer, to eliminate problems with uninitialized pointers
	Error:= TRUE;
	RETURN;
END_IF

thisloopstarttime:= TIME();	//store the time of the beginning of this loop
Done:= FALSE;
Execute_TRIG(CLK:= Execute);
Abort_TRIG(CLK:= Abort);

IF Execute_TRIG.Q THEN
//must see a rising edge on execute to start composing
	starttime:= TIME();	//store the time of the beginning of execution
	compose:= TRUE;
	Busy:= TRUE;
	Aborted:= FALSE;
	//need to init every sing struct at first time...
	lastindex:= MIN(NumberOfVars, GPL_JSON.MAX_VARS);
	IF NOT JSONVars^[1].Init THEN
		JSONVars^[1].Init := Init();
	END_IF
	
	Error:= FALSE;
	ErrorPosition:= 0;
	bufferposition:= 1;
	jsonvarindex:= 1;
	objectLevel := 0;	
	FOR i:= 1 TO GPL_JSON.MAX_LEVELS DO
	//clear names array
		names[i].Name:= '';
		names[i].ArrayIndex:= 0;
	END_FOR
	//clear previous string
	SysMemSet(
		pDest:= JSONString, 
		udiValue:= 0, 
		udiCount:= JSONStringSize
	);
END_IF

IF Abort_TRIG.Q THEN
	Busy:= FALSE;
	Aborted:= TRUE;
	compose:= FALSE;
END_IF

WHILE compose AND (jsonvarindex <= lastindex) AND (bufferposition < JSONStringSize) DO 
//loop through all variables

	names:= JSONVars^[jsonvarindex].Names;	//helper variable for name array property

	IF (jsonvarindex = 1) THEN
	//first object, no comma
		objectstr:= '{';	//new JSON string	
		IF Format THEN
			objectstr:= CONCAT(objectstr, GPL_JSON.NEWLINE);
		END_IF
	ELSE
		objectstr:= '';	//clear previous object string	
		IF NOT (VariableArraySize AND (names[1].ArrayIndex > 0) AND (JSONVars^[jsonvarindex].ValueType = JSONVALUETYPE.json_null)) THEN
		//don't write the value if the current variable is an array, and the value is null
			objectstr:= CONCAT(objectstr, ',');	//comma in between each value
			IF Format AND (names[1].ArrayIndex <= 1) THEN
			//new line after each comma, except in arrays
				objectstr:= CONCAT(objectstr, GPL_JSON.NEWLINE);	
			END_IF	
		END_IF
	END_IF

	IF (MaxLevel = 0) THEN
	//default, create all objects below the program level
		maxlevelindex:= JSONVars^[jsonvarindex].ApplicationLevel - 2;
	ELSE
	//manually defined with the MaxLevel input
		IF (jsonvarindex = 1) THEN
			maxlevelindex:= MaxLevel;
		ELSE
			maxlevelindex:= JSONVars^[jsonvarindex].ApplicationLevel - 2;	
		END_IF
	END_IF
	
	FOR namesindex:= maxlevelindex TO 1 BY -1 DO 
	//loop through all levels of an object in reverse
		//======================open new objects or arrays, or create new name:value pairs======================
		IF names[namesindex].NewArray AND (names[namesindex].ArrayIndex <= 1) THEN
		//new array at this level
			CreateName(Name:= names[namesindex].Name);
			CreateArray();
		END_IF	
		IF names[namesindex].NewObject AND (namesindex <> 1) THEN
		//new object at this level
			IF (NOT inArray) THEN
				CreateName(Name:= names[namesindex].Name);
			END_IF	
			CreateObject();		
		END_IF
		
		IF (namesindex=1) THEN
		//only write a value at level 1
			IF (names[namesindex].ArrayIndex > 0) THEN
			//array, create value only
				IF NOT (VariableArraySize AND (names[1].ArrayIndex > 0) AND (JSONVars^[jsonvarindex].ValueType = JSONVALUETYPE.json_null)) THEN
				//don't write the value if the current variable is an array, and the value is null
					CreateValue(ValueType:= JSONVars^[jsonvarindex].ValueType, Value:= JSONVars^[jsonvarindex].AsString);					
				END_IF
			ELSE
			//name:value pair
				CreateName(Name:= names[namesindex].Name);
				CreateValue(ValueType:= JSONVars^[jsonvarindex].ValueType, Value:= JSONVars^[jsonvarindex].AsString);
			END_IF
		END_IF
	END_FOR
	
	
	IF (MaxLevel = 0) THEN
	//default, close all objects below the program level
		closeLevel:= JSONVars^[jsonvarindex].ApplicationLevel - 2;
	ELSE
	//manually defined with the MaxLevel input
		IF jsonvarindex = 1 THEN
			closeLevel:= 1;
		ELSE
			closeLevel:= JSONVars^[jsonvarindex].ApplicationLevel - 2;	
		END_IF
	END_IF
	
	FOR namesindex:= 1 TO closeLevel DO 
	//start at the lowest level and count up
	//close objects or arrays if this is the last value in this object or array
		IF names[namesindex].EndObject AND (namesindex <> 1) THEN
		//close object at this level
			CloseObject();
		END_IF
		
		IF names[namesindex].EndArray THEN	
		//close array at this level
			CloseArray();	
		END_IF		
		
	END_FOR	
	
	//concatenate the temporary object string to the JSON string output
	StrConcatA(
		pstFrom:= ADR(objectstr), 
		pstTo:= ADR(JSONString^[bufferposition]), 
		iBufferSize:= UDINT_TO_INT(JSONStringSize)
	);	
	
	bufferposition:= bufferposition + DINT_TO_UDINT(LEN(objectstr));

	IF (jsonvarindex >= NumberOfVars) THEN
	//end of vars, close string
		compose:= FALSE;
		Busy:= FALSE;
		Done:= TRUE;		
		ComposeTime:= TIME() - starttime;
		JSONString^[bufferposition]:= ASCII.CLOSE_BRACE;;	//close JSON object with }
		bufferposition:= bufferposition + 1;
		JSONString^[bufferposition]:= ASCII.NULL;	//null character to end string
	END_IF
	
	IF TIME() >= (thisloopstarttime + GPL_JSON.MAX_EXECUTION_TIME) THEN
	//this function block won't take up more than GPL_JSON.MAX_EXECUTION_TIME on one scan
	//very long strings could take too long to compose in one task cycle, and cause a watchdog exception
		RETURN;
	END_IF
	
	jsonvarindex:= jsonvarindex + 1;	
END_WHILE

(*
| Author: Tim Van Meppelen, Pro Electric Inc.
| timv@proelectric.com
| Date: Oct 22, 2018
| close a JSON array
*)
METHOD PRIVATE CloseArray
objectstr:= CONCAT(objectstr, ']');

IF Format THEN
	objectstr:= CONCAT(objectstr, GPL_JSON.NEWLINE);	
END_IF

inArray := FALSE;
END_METHOD

(*
| Author: Tim Van Meppelen, Pro Electric Inc.
| timv@proelectric.com
| Date: Oct 22, 2018
| close a JSON object
*)
METHOD PRIVATE CloseObject
VAR
	indent:		INT;
END_VAR
IF Format THEN
	FOR indent:= 1 TO JSONVars^[jsonvarindex].ApplicationLevel-1 DO
		objectstr:= CONCAT(objectstr, GPL_JSON.INDENT);	
	END_FOR
END_IF

IF objectLevel > 0 THEN
	objectstr:= CONCAT(objectstr, '}');
	objectLevel := objectLevel - 1;
END_IF
END_METHOD

(*
| Author: Tim Van Meppelen, Pro Electric Inc.
| timv@proelectric.com
| Date: Oct 22, 2018
| create a new JSON array
| 
| [ ------ ------------ value ---------------- ] 
|         /                               \
| 	      \_______________ , _____________/
| 		
*)
METHOD PRIVATE CreateArray
objectstr:= CONCAT(objectstr, '[');	//opening [

inArray := TRUE;
END_METHOD

(*
| Author: Tim Van Meppelen, Pro Electric Inc.
| timv@proelectric.com
| Date: Oct 22, 2018
| create a JSON name string from a local variable of type JSONVAR
*)
METHOD PRIVATE CreateName
VAR_INPUT
	Name:	 		STRING(GPL_JSON.MAX_NAME_SIZE);
END_VAR
VAR
	indent:			INT;
	leadingpos:		INT;
END_VAR
IF Format THEN
	FOR indent:= 1 TO JSONVars^[jsonvarindex].ApplicationLevel-1 DO
		objectstr:= CONCAT(objectstr, GPL_JSON.INDENT);	
	END_FOR
END_IF

objectstr:= CONCAT(objectstr, '"');	//opening quote

leadingpos:= FIND(Name, GPL_JSON.IGNORE_LEADING_CHAR);
//if leading character is configured and present, delete it from the name
IF (leadingpos = 1) THEN
	objectstr:= CONCAT(objectstr, DELETE(Name, 1, 1));//variable name
ELSE
	objectstr:= CONCAT(objectstr, Name);//variable name
END_IF

objectstr:= CONCAT(objectstr, '":');	//closing quote and name:value separator
END_METHOD

(*
| Author: Tim Van Meppelen, Pro Electric Inc.
| timv@proelectric.com
| Date: Oct 22, 2018
| create a new JSON object
| 
| {------ "name" ------ : ----- value --------- }
|     /                                 \
| 	  \_______________ , _______________/
| 
*)
METHOD PRIVATE CreateObject
objectstr:= CONCAT(objectstr, '{');	//opening {

IF Format THEN
	objectstr:= CONCAT(objectstr, GPL_JSON.NEWLINE);
END_IF

objectLevel := objectLevel + 1;
END_METHOD

(*
| Author: Tim Van Meppelen, Pro Electric Inc.
| timv@proelectric.com
| Date: Oct 22, 2018
| create a JSON value string from a local variable of type JSONVAR
*)
METHOD PRIVATE CreateValue
VAR_INPUT
	ValueType:		JSONVALUETYPE;
	Value:			STRING(GPL_JSON.MAX_VALUE_SIZE);
END_VAR
CASE ValueType OF
//append value to object string
JSONVALUETYPE.json_number:
	objectstr:= CONCAT(objectstr, Value);
JSONVALUETYPE.json_integer:
	objectstr:= CONCAT(objectstr, Value);	
JSONVALUETYPE.json_boolean:
	objectstr:= CONCAT(objectstr, Value);
JSONVALUETYPE.json_string:
	objectstr:= CONCAT(objectstr, '"');	//opening quote
	objectstr:= CONCAT(objectstr, Value);
	objectstr:= CONCAT(objectstr, '"');	//closing quote
JSONVALUETYPE.json_null:
	objectstr:= CONCAT(objectstr, 'null');
END_CASE
END_METHOD

(*
| Author: Tim Van Meppelen, Pro Electric Inc.
| timv@proelectric.com
| Date: Oct 22, 2018
| Something went wrong, return the index of the variable where the problem was encountered
*)
METHOD PRIVATE ErrorHandler
compose:= FALSE;
Busy:= FALSE;
Error:= TRUE;
ErrorPosition:= jsonvarindex;	//return buffer position of unexpected character
RETURN;
END_METHOD

METHOD PRIVATE Init : BOOL
VAR
	varlevelindex:		INT;
END_VAR
//======================Set first and lastvariable properties======================
//characteristics of the first and last variable are not always set properly by FB_Init
FOR varlevelindex:= 1 TO JSONVars^[1].ApplicationLevel-2 DO
//every level of the first variable could be either a new object or a new array
	IF (JSONVars^[1].Names[varlevelindex].ArrayIndex = 1) THEN
	//new array at the first array object
		JSONVars^[1].Names[varlevelindex].NewArray:= TRUE;	
	ELSIF (varlevelindex > 1) OR (NumberofVars = 1) THEN
	//new object at every level, special case for single variables
		JSONVars^[1].Names[varlevelindex].NewObject:= TRUE;
	END_IF			
END_FOR

//lastindex:= MIN(NumberOfVars, GPL_JSON.MAX_VARS);
FOR varlevelindex:= 1 TO JSONVars^[lastindex].ApplicationLevel-2 DO
//close all open arrays and objects
	IF (JSONVars^[lastindex].Names[varlevelindex].ArrayIndex > 0) THEN
	//end array if an array index exists
		JSONVars^[lastindex].Names[varlevelindex].EndArray:= TRUE;	
	ELSIF (varlevelindex > 1) OR (NumberofVars = 1) THEN
	//end all objects, special case for single variables
		JSONVars^[lastindex].Names[varlevelindex].EndObject:= TRUE;
	END_IF			
END_FOR

Init:= TRUE;
END_METHOD

END_FUNCTION_BLOCK

// Functions/JSONVALUE_TO_STRING
(*
| Author: Tim Van Meppelen, Pro Electric Inc.
| timv@proelectric.com
| Date: May 4, 2021
| convert a JSON value to string
*)
FUNCTION JSONVALUE_TO_STRING : STRING
VAR_INPUT
	In_JSON:		POINTER TO JSONVAR;
END_VAR

CASE In_JSON^.ValueType OF
JSONVALUETYPE.json_null:
	JSONVALUE_TO_STRING:= 'null';
JSONVALUETYPE.json_boolean:
	IF In_JSON^.Boolean THEN
		JSONVALUE_TO_STRING:= 'true';
	ELSE
		JSONVALUE_TO_STRING:= 'false';
	END_IF
JSONVALUETYPE.json_number:
	JSONVALUE_TO_STRING:= REAL_TO_STRING_X(In_JSON^.Number);
JSONVALUETYPE.json_integer:
	JSONVALUE_TO_STRING:= DINT_TO_STRING(In_JSON^.Integer);
JSONVALUETYPE.json_string:
	JSONVALUE_TO_STRING:= In_JSON^.CharString;
END_CASE

END_FUNCTION

// Functions/REAL_TO_STRING_X
(*
| Author: Tim Van Meppelen, Pro Electric Inc.
| timv@proelectric.com
| Date: Nov 2, 2018
| Standard REAL_TO_STRING function will always add a decimal place even if the input is a whole number
| this function will drop the ".0" on the string output
*)
FUNCTION REAL_TO_STRING_X : STRING
VAR_INPUT
	In_REAL:		REAL;
END_VAR
VAR
	TempVar:		STRING;
END_VAR

TempVar:= REAL_TO_STRING(In_REAL);
IF (RIGHT(STR:= TempVar, SIZE:= 2) = '.0') THEN
	REAL_TO_STRING_X:= DELETE(STR:= TempVar, LEN:= 2, POS:= LEN(TempVar) - 1);
ELSE
	REAL_TO_STRING_X:= TempVar;
END_IF

END_FUNCTION

// Functions/STRING_TO_JSONVALUE
(*
| Author: Tim Van Meppelen, Pro Electric Inc.
| timv@proelectric.com
| Date: May 4, 2021
| Convert a string to a JSON value
*)
FUNCTION STRING_TO_JSONVALUE
VAR_INPUT
	In_String:		STRING;
	Out_JSON:		POINTER TO JSONVAR;
END_VAR
VAR
	TempBool:	BOOL;
	TempReal:	REAL;
	TempInt:	DINT;
	TempString:	STRING(255);
END_VAR

IF (Out_JSON^.ValueType = JSONVALUETYPE.json_null) THEN
//if the type is not explicitly configured, make a guess at the type
	IF ISINTEGER(ADR(In_String)) THEN
		Out_JSON^.ValueType:= JSONVALUETYPE.json_integer;
	ELSIF ISNUMBER(ADR(In_String)) THEN
		Out_JSON^.ValueType:= JSONVALUETYPE.json_number;
	ELSIF ISBOOLEAN(ADR(In_String)) THEN
		Out_JSON^.ValueType:= JSONVALUETYPE.json_boolean;
	ELSIF (In_String = 'null') THEN
		Out_JSON^.ValueType:= JSONVALUETYPE.json_null;
	ELSE
		Out_JSON^.ValueType:= JSONVALUETYPE.json_string;
	END_IF
END_IF

CASE Out_JSON^.ValueType OF
JSONVALUETYPE.json_null:
	Out_JSON^.Null:= 'null';
JSONVALUETYPE.json_boolean:
	StrToUpperA(pString:= ADR(In_String));
	IF (In_String = 'TRUE') THEN
		TempBool:= TRUE;
	ELSE
		TempBool:= FALSE;
	END_IF
	Out_JSON^.Boolean:= TempBool;
JSONVALUETYPE.json_integer:
	TempInt:= STRING_TO_DINT(In_String);
	Out_JSON^.Integer:= TempInt;	
JSONVALUETYPE.json_number:
	TempReal:= STRING_TO_REAL(In_String);
	Out_JSON^.Number:= TempReal;
JSONVALUETYPE.json_string:
	Out_JSON^.CharString:= In_String;
END_CASE

END_FUNCTION

// Functions/ISINTEGER
(*
| Author: Tim Van Meppelen, Pro Electric Inc.
| timv@proelectric.com
| Date: Mar 2, 2020
| check if a string contains an integer, allows for "-" at the beginning of the string, and no decimals
*)
FUNCTION ISINTEGER : BOOL
VAR_INPUT
	In:		POINTER TO ARRAY[1..255] OF BYTE;
END_VAR
VAR
	i:				UINT;
	founddecimal:	BOOL;
END_VAR

FOR i:= 1 TO 255 DO
	CASE In^[i] OF 	
	ASCII.NULL:
	//end of string
		EXIT;
	ASCII.MINUS:
	//only allow a "-" in the first position	
		IF (i=1) THEN
			ISINTEGER:= TRUE;
		ELSE
			ISINTEGER:= FALSE;
			EXIT;
		END_IF
	ASCII.DOT:
	//no decimal points allowed in integers
		ISINTEGER:= FALSE;
		EXIT;
	ASCII.NUMBER_0..ASCII.NUMBER_9:
		ISINTEGER:= TRUE;
	ELSE
	//all other characters are not part of numbers
		ISINTEGER:= FALSE;
		EXIT;
	END_CASE
END_FOR

END_FUNCTION

// Functions/ISNUMBER
(*
| Author: Tim Van Meppelen, Pro Electric Inc.
| timv@proelectric.com
| Date: Oct 2, 2018
| check if a string contains a valid number, allows for "-" at the beginning of the string, and one "." character
*)
FUNCTION ISNUMBER : BOOL
VAR_INPUT
	In:		POINTER TO ARRAY[1..255] OF BYTE;
END_VAR
VAR
	i:				UINT;
	founddecimal:	BOOL;
END_VAR

FOR i:= 1 TO 256 DO
	CASE In^[i] OF 	
	ASCII.NULL:
	//end of string
		RETURN;
	ASCII.MINUS:
	//only allow a "-" in the first position	
		IF (i=1) THEN
			ISNUMBER:= TRUE;
		ELSE
			ISNUMBER:= FALSE;
			RETURN;
		END_IF
	ASCII.DOT:
	//only allow one decimal point
		IF founddecimal THEN
		//already found one decimal, can't have two
			ISNUMBER:= FALSE;
			RETURN;
		ELSE
		//first decimal point found, allow one
			ISNUMBER:= TRUE;
			founddecimal:= TRUE;
		END_IF
	ASCII.NUMBER_0..ASCII.NUMBER_9:
		ISNUMBER:= TRUE;
	ELSE
	//all other characters are not part of numbers
		ISNUMBER:= FALSE;
		RETURN;
	END_CASE
END_FOR

END_FUNCTION

// Functions/ISBOOLEAN
(*
| Author: Tim Van Meppelen, Pro Electric Inc.
| timv@proelectric.com
| Date: Oct 2, 2018
| check if a string would convert to a valid boolean variable
*)
FUNCTION ISBOOLEAN : BOOL
VAR_INPUT
	In:		POINTER TO STRING(5);
END_VAR
VAR
	TempVar:	STRING(5);
END_VAR

TempVar:= In^;
StrToUpperA(pString:= ADR(TempVar));

ISBOOLEAN:= (TempVar = 'TRUE') OR (TempVar = 'FALSE');

END_FUNCTION

// Functions/SPLIT_VARNAME
(*
| Author: Tim Van Meppelen, Pro Electric Inc.
| timv@proelectric.com
| Date: June 26, 2018
| split a string into an array at the '.' character
| modified from https://forum.codesys.com/viewtopic.php?t=9889
| 'a.b.c.d' becomes an array[1]=d, [2]=c, [3]=b, [4]=a
*)
FUNCTION SPLIT_VARNAME : UINT;
VAR_INPUT
	VarNameArray:	REFERENCE TO ARRAY[1..GPL_JSON.MAX_LEVELS] OF JSONVARNAME;
	StringIn: 		STRING(GPL_JSON.MAX_VAR_NAME);	//input string
END_VAR

VAR CONSTANT
	SPLIT_CHAR : 	STRING(1):= '.';	
END_VAR

VAR
	ArraySize:			UINT:= 1;
    sShortString : 		STRING;
    iSplitLocation : 	INT;
	i:					UINT;
	TempArray:			ARRAY[1..GPL_JSON.MAX_LEVELS] OF STRING;
END_VAR

//Loop through string until there is no string left or array has hit its limits
WHILE (StrLenA(pstData:= ADR(StringIn)) > 0) DO
	//Find location of first break point
	iSplitLocation := StrFindA(
		pst1:= ADR(StringIn), 
		pst2:= ADR(SPLIT_CHAR), 
		uiSearchStart:= 1
	) - 1;
	
	//If there is no break point found then set location to size of string
	IF (iSplitLocation = -1) THEN
		iSplitLocation := DINT_TO_INT(StrLenA(pstData:= ADR(StringIn)));
	END_IF
  
	//Copy the part of the string that is needed for the parameter.
	StrMidA(
		pst:= ADR(StringIn), 
		uiInputBufferSize:= SIZEOF(StringIn), 
		iLength:= iSplitLocation, 
		iPosition:= 1, 
		pstResult:= ADR(sShortString), 
		uiResultBufferSize:= SIZEOF(sShortString)
	);

	//Make sure string is not empty before using up an array spot.
	IF (StrLenA(pstData:= ADR(sShortString)) > 0) THEN
		TempArray[ArraySize] := sShortString;
		ArraySize := ArraySize + 1;
	END_IF

	//Remove copied components from long string
	StrDeleteA(
		pby:= ADR(StringIn), 
		iLength:= (iSplitLocation + LEN(SPLIT_CHAR)), 
		iPosition:= 1
	);

	//Check to see if more parameters can fit in array. If not exit loop
	IF (ArraySize > GPL_JSON.MAX_LEVELS) THEN
		EXIT;
	END_IF 
END_WHILE

ArraySize:= ArraySize - 1;

FOR i:= 0 TO ArraySize DO
//reverse the order of the array
	VarNameArray[i+1].Name:= TempArray[ArraySize-i];	
END_FOR

SPLIT_VARNAME:= ArraySize;

END_FUNCTION

// Examples/ExampleJSON_PRG
(*
| Author: Tim Van Meppelen, Pro Electric Inc.
| timv@proelectric.com
| Date: Nov 2, 2018
| example program demonstrating JSONVAR, STRUCT_TO_JSON, AND JSON_TO_STRUCT
| 
| This example will populate a structure with values and types.  On a rising edge of ComposeJSON.Execute, 
| ComposeJSON will create a JSON string.  When ComposeJSON.Done is set, ParseJSON.Execute is set, and 
| ParseJSON will then parse that string back into a different structure.
*)
PROGRAM ExampleJSON_PRG
VAR
	LocalJSONObj:		EXAMPLEJSONSTRUCT;
	ComposeJSON:		STRUCT_TO_JSON;
	
	JSONString:			STRING(1000);

	NewJSONObj:			EXAMPLEJSONSTRUCT;	
	ParseJSON:			JSON_TO_STRUCT;
	
	CreateJSONInFB:		EXAMPLE_FB;
END_VAR

LocalJSONObj.var1.Boolean:= TRUE;
LocalJSONObj.var2.Number:= 34.8756;
LocalJSONObj.var3.CharString:= 'teststring';
LocalJSONObj.obj.var4.Number:= 22;
LocalJSONObj.obj.var5.AsString:= 'FALSE';	//JSONVAR will guess at type, in this case, boolean
LocalJSONObj.obj.var6.CharString:= 'qwer';
LocalJSONObj.obj.var7[1].Number:= 123.234;
LocalJSONObj.obj.var7[2].AsString:= '55.46';	//JSONVAR will guess at type, in this case, a number
LocalJSONObj.obj.var7[3].Number:= 985;
LocalJSONObj.arrayobj[1].Number:= 1;
LocalJSONObj.arrayobj[2].Number:= 2;
LocalJSONObj.arrayobj[3].Number:= 3;

//create a JSON string from local object
ComposeJSON(
	JSONString:= ADR(JSONString), 
	JSONStringSize:= SIZEOF(JSONString),
	JSONVars:= ADR(LocalJSONObj),
	NumberOfVars:= SIZEOF(LocalJSONObj) / SIZEOF(JSONVAR)
);

//fill another local object with values from the created JSON string
ParseJSON(
	Execute:= ComposeJSON.Done,
	JSONString:= ADR(JSONString), 
	JSONStringSize:= SIZEOF(JSONString),
	JSONVars:= ADR(NewJSONObj),
	NumberOfVars:= SIZEOF(NewJSONObj) / SIZEOF(JSONVAR)
);

CreateJSONInFB();

END_PROGRAM

// Examples/EXAMPLE_FB
(*
| Author: Tim Van Meppelen, Pro Electric Inc.
| timv@proelectric.com
| Date: Jan 31, 2020
| example of use in a function block
*)
FUNCTION_BLOCK EXAMPLE_FB
VAR_INPUT
	MaxLevel:			INT;
END_VAR
VAR_OUTPUT
	Out:				STRING(255);
END_VAR
VAR
	color_temp:			JSONVAR;
	FirstScan:			BOOL:= TRUE;
	ComposeJSON:		STRUCT_TO_JSON;
END_VAR

color_temp.CharString:= 'red';

ComposeJSON(
	JSONString:= ADR(Out), 
	JSONStringSize:= SIZEOF(Out),
	JSONVars:= ADR(color_temp),
	NumberOfVars:= SIZEOF(color_temp) / SIZEOF(JSONVAR),
	MaxLevel:= MaxLevel
);

IF FirstScan THEN
	FirstScan:= FALSE;
	ComposeJSON.Execute:= TRUE;
END_IF

END_FUNCTION_BLOCK

// Functions/CLEANSTRING
(*
| Author: Tim Van Meppelen, Pro Electric Inc.
| timv@proelectric.com
| Date: Oct 9, 2018
| strip all control characters and spaces from a string
*)
FUNCTION CLEANSTRING : BOOL
VAR_INPUT
	StringPtr:		POINTER TO ARRAY[1..MAXSTRINGLENGTH] OF BYTE;
END_VAR
VAR CONSTANT
	MAXSTRINGLENGTH:	UINT:= 2048;
END_VAR
VAR
	i:				UINT;
	j:				UINT;
END_VAR

FOR i:= 1 TO MAXSTRINGLENGTH DO
	IF (StringPtr^[i] >= 1) AND (StringPtr^[i] <= 16#20) THEN
	//match all control and white space characters, except for null, which terminates a string
		FOR j:= i TO MAXSTRINGLENGTH DO
			IF (StringPtr^[j] = ASCII.NULL) THEN
			//null character terminates string
				EXIT;
			ELSE
			//shift character array left one
				StringPtr^[j]:= StringPtr^[j+1];
			END_IF
		END_FOR
		i:= i - 1;	//run loop at same position again
	ELSIF (StringPtr^[i] = ASCII.NULL) THEN
	//found null character at the end of the string
		EXIT;
	END_IF
END_FOR

CLEANSTRING:= TRUE;

END_FUNCTION

// Examples/Test_ArrayOfStruct_PRG
PROGRAM Test_ArrayOfStruct_PRG
VAR
	FirstScan:			BOOL:= TRUE;	
	
	LocalJSONObj:		ARRAYOFSTRUCT;
	ComposeJSON:		STRUCT_TO_JSON;
	JSONString:			STRING(255);

END_VAR

IF FirstScan THEN
	FirstScan:= FALSE;
	ComposeJSON.Execute:= TRUE;
END_IF

//create a JSON string
LocalJSONObj.arr[1].obj1.Number:= 23.5;
LocalJSONObj.arr[1]._obj2.Integer:= 3;
LocalJSONObj.arr[1].obj3.Boolean:= TRUE;

LocalJSONObj.arr[2].obj1.Number:= 54.5;
LocalJSONObj.arr[2]._obj2.Number:= 7.5;
LocalJSONObj.arr[2].obj3.Boolean:= FALSE;

LocalJSONObj.arr[3].obj1.Number:= 87.1;
LocalJSONObj.arr[3]._obj2.Integer:= 88;
LocalJSONObj.arr[3].obj3.Boolean:= TRUE;

LocalJSONObj.arr[4].obj1.Boolean:= FALSE;
LocalJSONObj.arr[4]._obj2.Number:= 132.55;
LocalJSONObj.arr[4].obj3.Integer:= 3;


ComposeJSON(
	JSONString:= ADR(JSONString), 
	JSONStringSize:= SIZEOF(JSONString),
	JSONVars:= ADR(LocalJSONObj),
	NumberOfVars:= SIZEOF(LocalJSONObj) / SIZEOF(JSONVAR)
);

END_PROGRAM

// Examples/Test_Array_PRG
PROGRAM Test_Array_PRG
VAR
	FirstScan:			BOOL:= TRUE;	
	
	testarray:			ARRAY[1..20] OF JSONVAR;
	ComposeJSON:		STRUCT_TO_JSON;
	JSONString:			STRING(255);
	
	NewString:			STRING(255):= '{"new":["234","34.5","98.4","10.4","812","5","23","65","95.6","98","234","34.5","98.4","10.4","812","5","23","65","95.6","98"]}';
	ParseJSON:			JSON_TO_STRUCT;
	new:				ARRAY[1..20] OF JSONVAR;	
END_VAR

IF FirstScan THEN
	FirstScan:= FALSE;
	ComposeJSON.Execute:= TRUE;
	ParseJSON.Execute:= TRUE;
END_IF

//create a JSON string
testarray[1].Number:= 32.5;
testarray[2].Number:= 65.2;
testarray[3].Number:= 81.54;
testarray[4].Number:= 1953.523;
testarray[5].Number:= 901.5;

ComposeJSON(
	JSONString:= ADR(JSONString), 
	JSONStringSize:= SIZEOF(JSONString),
	JSONVars:= ADR(testarray),
	NumberOfVars:= SIZEOF(testarray) / SIZEOF(JSONVAR)
);




//parse a JSON string and put it into a variable
ParseJSON(
	JSONString:= ADR(NewString), 
	JSONStringSize:= SIZEOF(NewString),
	JSONVars:= ADR(new),
	NumberOfVars:= SIZEOF(new) / SIZEOF(JSONVAR)
);

END_PROGRAM

// Examples/Test_NestedStruct_PRG
PROGRAM Test_NestedStruct_PRG
VAR
	FirstScan:			BOOL:= TRUE;	
	
	LocalJSONObj:		JSONSTRUCT_1;
	ComposeJSON:		STRUCT_TO_JSON;
	JSONString:			STRING(255);
	
	NewString:			STRING(255):= '{"new":{"obj1":"234", "obj2":"34.5", "obj3":"true","nest":{"obj1":"468.5", "obj2":"197", "obj3":"this is a string"}}}';
	ParseJSON:			JSON_TO_STRUCT;
	new:				JSONSTRUCT_1;
END_VAR

IF FirstScan THEN
	FirstScan:= FALSE;
	ComposeJSON.Execute:= TRUE;
	ParseJSON.Execute:= TRUE;
END_IF

//create a JSON string
LocalJSONObj.obj1.Number:= 23.5;
LocalJSONObj.obj2.Integer:= 3;
LocalJSONObj.obj3.Boolean:= TRUE;

ComposeJSON(
	JSONString:= ADR(JSONString), 
	JSONStringSize:= SIZEOF(JSONString),
	JSONVars:= ADR(LocalJSONObj),
	NumberOfVars:= SIZEOF(LocalJSONObj) / SIZEOF(JSONVAR)
);





//parse a JSON string and put it into a variable
ParseJSON(
	JSONString:= ADR(NewString), 
	JSONStringSize:= SIZEOF(NewString),
	JSONVars:= ADR(new),
	NumberOfVars:= SIZEOF(new) / SIZEOF(JSONVAR)
);

END_PROGRAM

// Examples/Test_SingleVar_PRG
PROGRAM Test_SingleVar_PRG
VAR
	FirstScan:			BOOL:= TRUE;	
	
	colour:				JSONVAR;	
	ComposeJSON:		STRUCT_TO_JSON;
	JSONString:			STRING(255);
	
	NewString:			STRING:= '{"color":"blue"}';
	ParseJSON:			JSON_TO_STRUCT;
	color:				JSONVAR;
END_VAR

IF FirstScan THEN
	FirstScan:= FALSE;
	ComposeJSON.Execute:= TRUE;
	ParseJSON.Execute:= TRUE;
END_IF

//create a JSON string from a variable
colour.CharString:= 'blue';
ComposeJSON(
	JSONString:= ADR(JSONString), 
	JSONStringSize:= SIZEOF(JSONString),
	JSONVars:= ADR(colour),
	NumberOfVars:= SIZEOF(colour) / SIZEOF(JSONVAR)
);



//parse a JSON string and put it into a variable
ParseJSON(
	JSONString:= ADR(NewString), 
	JSONStringSize:= SIZEOF(NewString),
	JSONVars:= ADR(color),
	NumberOfVars:= SIZEOF(color) / SIZEOF(JSONVAR)
);

END_PROGRAM

// Examples/Test_Struct_PRG
PROGRAM Test_Struct_PRG
VAR
	FirstScan:			BOOL:= TRUE;	
	
	LocalJSONObj:		JSONSTRUCT;
	ComposeJSON:		STRUCT_TO_JSON;
	JSONString:			STRING(255);
	
	NewString:			STRING:= '{"new":{"obj1":"234", "_obj2":"34.5", "obj3":"true"}}';
	ParseJSON:			JSON_TO_STRUCT;
	new:				JSONSTRUCT;
END_VAR

IF FirstScan THEN
	FirstScan:= FALSE;
	ComposeJSON.Execute:= TRUE;
	ParseJSON.Execute:= TRUE;
END_IF

//create a JSON string
LocalJSONObj.obj1.Number:= 23.5;
LocalJSONObj._obj2.Integer:= 3;
LocalJSONObj.obj3.Boolean:= TRUE;

ComposeJSON(
	JSONString:= ADR(JSONString), 
	JSONStringSize:= SIZEOF(JSONString),
	JSONVars:= ADR(LocalJSONObj),
	NumberOfVars:= SIZEOF(LocalJSONObj) / SIZEOF(JSONVAR)
);



//parse a JSON string and put it into a variable
ParseJSON(
	JSONString:= ADR(NewString), 
	JSONStringSize:= SIZEOF(NewString),
	JSONVars:= ADR(new),
	NumberOfVars:= SIZEOF(new) / SIZEOF(JSONVAR)
);

END_PROGRAM
